PROGRAM UN01_StateMachineBox
VAR
	FB_StateMachineShorting	: FB_StateManager;
END_VAR

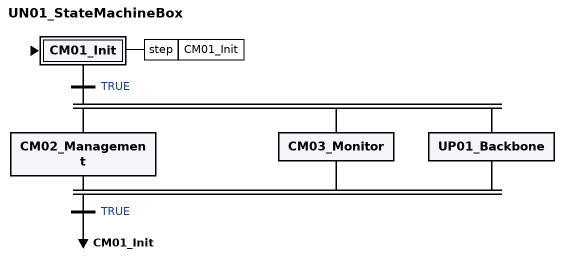
INITIAL_STEP CM01_Init:
    CM01_Init(N);  // step action
END_STEP
TRANSITION FROM CM01_Init TO (CM02_Management, CM03_Monitor, UP01_Backbone)
    := TRUE;
END_TRANSITION
STEP CM02_Management:
END_STEP
STEP CM03_Monitor:
END_STEP
STEP UP01_Backbone:
END_STEP
TRANSITION FROM (CM02_Management, CM03_Monitor, UP01_Backbone) TO CM01_Init
    := TRUE;
END_TRANSITION

ACTION CM01_Init:
//Shorting
Data_GVL.bFL_StartShorting 			:= Data_GVL.bStartButton OR HMI_GVL.bStartButtonShorting;
Data_GVL.bFL_StopShorting 			:= Data_GVL.bStopButton OR HMI_GVL.bStopButtonShorting;
Data_GVL.bFL_ResetShorting 			:= Data_GVL.bResetButton OR HMI_GVL.bResetButtonShorting;
Data_GVL.bFL_AutoManuaModeShorting 	:= NOT Data_GVL.StateMachineShorting.Running AND HMI_GVL.bTestModeEnableShorting;
END_ACTION

ACTION CM02_Management:
// NETWORK 1
END_ACTION

ACTION CM03_Monitor:
// NETWORK 1
END_ACTION

ACTION UP01_Backbone:
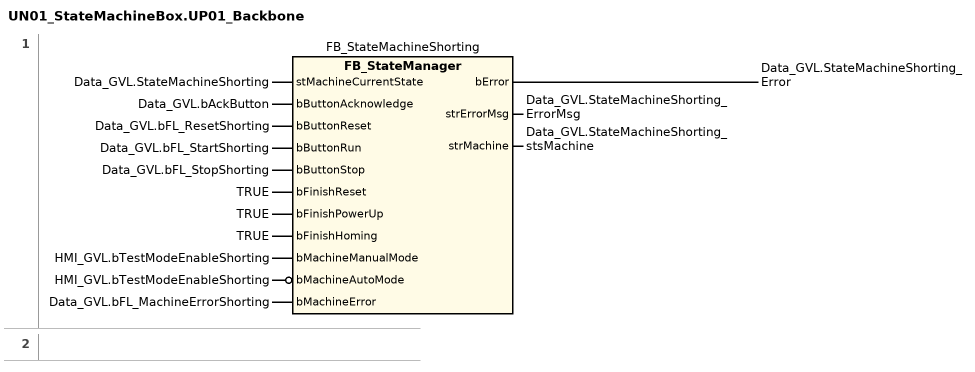
// NETWORK 1
FB_StateMachineShorting(
    stMachineCurrentState := Data_GVL.StateMachineShorting,
    bButtonAcknowledge := Data_GVL.bAckButton,
    bButtonReset := Data_GVL.bFL_ResetShorting,
    bButtonRun := Data_GVL.bFL_StartShorting,
    bButtonStop := Data_GVL.bFL_StopShorting,
    bFinishReset := TRUE,
    bFinishPowerUp := TRUE,
    bFinishHoming := TRUE,
    bMachineManualMode := HMI_GVL.bTestModeEnableShorting,
    bMachineAutoMode := NOT HMI_GVL.bTestModeEnableShorting,
    bMachineError := Data_GVL.bFL_MachineErrorShorting,
    strErrorMsg => Data_GVL.StateMachineShorting_ErrorMsg,
    strMachine => Data_GVL.StateMachineShorting_stsMachine); // FB_StateManager
Data_GVL.StateMachineShorting_Error := FB_StateMachineShorting.bError;

// NETWORK 2
END_ACTION

END_PROGRAM

(* stored: Version 1.1.0.1, ProductVersion 3.1.4024.9
   POU UN01_StateMachineBox: Id {7bfd295d-b76d-4d6b-a17a-998784b1a105}, SpecialFunc None
   Action CM01_Init: Id {a0ce267e-8ab5-4033-9e35-a07c9e761785}
   Action CM02_Management: Id {990c7f9a-b6ca-4207-9220-0dc81749c530}
   Action CM03_Monitor: Id {b1ba87fa-9ee2-4316-b6f7-e7c028a0b885}
   Action UP01_Backbone: Id {9f2aa1cf-e51e-4faf-8705-6d2d06f7aa6b} *)
